Staubli VAL3: SetProerty.pgx

public program SetProerty(string x_sTitle (dimensions=1), num x_nTopX (dimensions=1), num x_nTopY (dimensions=1), num x_nBottomX (dimensions=1), num x_nBottomY (dimensions=1), string& x_sListItem[] (dimensions=1), string& x_sItem (dimensions=1))
  local num l_nKey
  local num l_nItem
  local string l_sItem
begin
  //
  l_sItem=x_sItem
  call setSizeList(x_nTopX,x_nTopY,x_nBottomX,x_nBottomY)
  call listcreate(x_sTitle)
  call listadd(x_sListItem)
  call listupdate(0)
  call clear(0,13)
  call typeMenu(1,"OK")
  do
    l_nKey=getKey()
    call listevent(l_nKey,l_nItem,x_sItem)
    delay(0)
  until l_nKey==271 or l_nKey==270 or l_nKey==255
  if l_nKey==255
    x_sItem=l_sItem
  endIf
end
